(* IEC 61131-3 sources: myCodes/Stone/07.02.2022 - OOPs Approach/MPx_One_New/Mpx_One_Source_Code/MPx_One/3. USHPXMPX010A1/USHPXMPX010A1/MPXone_Medium/DFR_Libs (part 2) *)

/// Light Function ///

FUNCTION_BLOCK DFR_DiagLights
    VAR_INPUT
        Inp : BOOL;
        TotTime : REAL;
    END_VAR
    VAR_OUTPUT
        Out : BOOL;
        TimerDone : BOOL;
    END_VAR
    VAR
        LightTimer : DFRTimer;
    END_VAR
    IF Inp THEN
        LightTimer(Ena := Inp, PLCCycletime := 0.5, ProgramTime := TotTime);
        IF LightTimer.ElapsedTime <= (TotTime / 10) THEN
            Out := TRUE;
        ELSIF LightTimer.ElapsedTime > (TotTime / 10) AND LightTimer.ElapsedTime <= (TotTime / 7.5) THEN
            Out := FALSE;
        ELSIF LightTimer.ElapsedTime > (TotTime / 7.5) AND LightTimer.ElapsedTime <= (TotTime / 5) THEN
            Out := TRUE;
        ELSIF LightTimer.ElapsedTime > (TotTime / 5) AND LightTimer.ElapsedTime <= (TotTime / 2.5) THEN
            Out := FALSE;
        ELSIF LightTimer.ElapsedTime > (TotTime / 2.5) AND LightTimer.ElapsedTime <= (TotTime / 2) THEN
            Out := TRUE;
        ELSIF LightTimer.ElapsedTime > (TotTime / 2) AND LightTimer.ElapsedTime <= (TotTime / 1.5) THEN
            Out := FALSE;
        ELSIF LightTimer.ElapsedTime > (TotTime / 1.5) AND LightTimer.ElapsedTime <= (TotTime / 1.25) THEN
            Out := TRUE;
        ELSE
            Out := FALSE;
        END_IF;
        IF LightTimer.Q THEN
            LightTimer(Ena := FALSE);
            TimerDone := TRUE;
        END_IF;
    ELSE
        Out := FALSE;
        TimerDone := FALSE;
        LightTimer(Ena := FALSE);

    END_IF;
END_FUNCTION_BLOCK

/// ************  EOL Run Test Functions ************///

/// EOL Pull Down Test Function ///

FUNCTION_BLOCK DFR_Feature_PullDownTest
    VAR_INPUT
        Enable             : BOOL; // To Enable the Regulation
        CycleTime          : REAL; // To change the Cycle Time of the Pull Down Test Function
        Preset_RegTime     : REAL; // Regulation Timer
        Preset_RegFailTime : REAL; // Regulation Fail Timer
        Preset_WaitTime    : REAL; // Regulation Wait Timer
        In1                : REAL; // Discharge Air Temp
        In2                : REAL; // Defrost Temp
        Reg_SP             : REAL; // Regulation Setpoint
        FanSP              : REAL; // Fan Setpoint
        FanHystSP          : REAL; // Fan Hysterisis SP

    END_VAR
    VAR
        Reg_Fail_Timer     : DFRTimer; // Enable the Fail Timer if Discharge Air Temp fails to meet the SP
        RegulationTimer    : DFRTimer; // Enable Regulation Timer to monitor Discharge Air temp

    END_VAR
    VAR_OUTPUT
        DFR_Regulation_Sts : STRING; // DFR Regulation Test Status
        Out1               : BOOL; // CDU Enable - V_OM_Solenoid_Flag
        Out2               : BOOL; // Fan Enable - V_OM_Fans_Flag
    END_VAR

    IF Enable AND (V_CSM_EOL_Test_Result = 0 OR V_CSM_EOL_Test_Result = 3) THEN
        Out1 := TRUE;
        IF In1 <= Reg_SP THEN
            RegulationTimer(Ena := TRUE, PLCCycletime := CycleTime, ProgramTime := Preset_RegTime);
            Reg_Fail_Timer(Ena := FALSE);
            IF RegulationTimer.Q THEN
                DFR_Regulation_Sts := 'PAS';
                RegulationTimer(Ena := FALSE);
            END_IF;
        ELSE
            Reg_Fail_Timer(Ena := TRUE, PLCCycletime := CycleTime, ProgramTime := Preset_RegFailTime);
            RegulationTimer(Ena := FALSE);
            IF Reg_Fail_Timer.Q THEN
                DFR_Regulation_Sts := 'FAL';
                Reg_Fail_Timer(Ena := FALSE);
            END_IF;
        END_IF;

        IF  (DFR_CINCaseSystemComponent(6) = 0) OR (DFR_CINCaseSystemComponent(9) = 2) THEN // No Door Case and MT Case
            Out2 := TRUE;
        ELSIF (NOT (DFR_CINCaseSystemComponent(6) = 0) AND (DFR_CINCaseSystemComponent(9) = 1)) THEN // LT Door Case Only
            IF In2 <= FanSP THEN // Fans will be turned On if Defrost Temp is less than Fan Setpoint
                Out2 := TRUE;
            ELSIF In2 > FanSP + FanHystSP THEN
                Out2 := FALSE;
            END_IF;
        ELSE
            Out2 := FALSE;
        END_IF;
    ELSIF (DFR_Regulation_Sts = 'FAL') OR(DFR_Regulation_Sts = 'PAS') THEN
        RegulationTimer(Ena := FALSE);
        Reg_Fail_Timer(Ena := FALSE);
    END_IF;
END_FUNCTION_BLOCK

/// Defrost Cycle Test Function  ///

FUNCTION_BLOCK DFR_Feature_DefrostCycleTest
    VAR_INPUT
        Enable : BOOL;       // To Enable the Defrost Cycle Test
        CycleTime : REAL;
        Preset_DefFailTime : REAL;
        In1 : REAL; // Defrost Termination Temperature OR Discharge Air Temp (If Defrost Probe is absent)
        SetPoint : REAL;  // Defrost Termination Temperature SP

    END_VAR
    VAR
        Def_Fail_Timer : DFRTimer; // Enable the Fail Timer if change in Defrost Term Temp fails to meet the SP
        TempDelta : REAL;
        PrevIn : REAL;
        SaveFlag : bool := FALSE;
    END_VAR

    VAR_OUTPUT
        DFR_DefrostCycle_Sts : STRING; // DFR Defrost Cycle Test Status
        Out1 : BOOL; // CDU Disable - V_OM_Solenoid_Flag
        Out2 : BOOL; // Defrost Enable - V_OM_Defrost_Flag
        Out3 : BOOL; // Fan Disable - V_OM_Fans_Flag
        Out4 : BOOL; // Drain Heater - V_OM_DrainHeat_Flag
    END_VAR

    Def_Fail_Timer(Ena := Enable, PLCCycletime := CycleTime, ProgramTime := Preset_DefFailTime);
    IF Enable AND (V_CSM_EOL_Test_Result = 0 OR V_CSM_EOL_Test_Result = 3) THEN
        IF(NOT SaveFlag) THEN
            SaveFlag := TRUE;
            //PrevIn := In1;
        //ELSE
            //TempDelta := (In1 - PrevIn); // Discharge Air Temp difference
        END_IF;

        Out2 := TRUE; // Defrost Should be Enabled
        Out1 := FALSE; // CDU should be Disabled
        IF Out2 AND NOT Out1 THEN
            IF In1 > Setpoint THEN
                Def_Fail_Timer(Ena := FALSE);
                DFR_DefrostCycle_Sts := 'PAS';
            ELSE
                ;
            END_IF;
        END_IF;

        IF Def_Fail_Timer.Q THEN
            DFR_DefrostCycle_Sts := 'FAL';
            Def_Fail_Timer(Ena := FALSE);
        END_IF;

        IF  (DFR_CINCaseSystemComponent(6) = 0) OR (DFR_CINCaseSystemComponent(9) = 2) THEN // No Door Case and MT Case
            Out3 := TRUE; // Fans are ON
            Out4 := FALSE; // Drain Heater are Disabled
        ELSIF (NOT (DFR_CINCaseSystemComponent(6) = 0) AND (DFR_CINCaseSystemComponent(9) = 1)) THEN // LT Door Case Only
            Out3 := FALSE; // Fans are OFF
            Out4 := TRUE; // Drain Heater are Enabled
        ELSE
            Out3 := FALSE; // Fans are OFF
            Out4 := FALSE; // Drain Heater are Disabled
        END_IF;
    ELSE
        PrevIn := In1;
        TempDelta := 0;
        SaveFlag := FALSE;
        DFR_DefrostCycle_Sts := 'NA';
        Def_Fail_Timer(Ena := FALSE);
    END_IF;

END_FUNCTION_BLOCK
/*
FUNCTION_BLOCK DFR_MOV_AVERAGE
    VAR_INPUT
        in_sample : real;
        in_count  : uint := 1; //It should be less than total no. of array samples
    END_VAR

    VAR
        array_real : ARRAY[1..64] OF real;
        sum        : real;
        index      : uint := 1;
    END_VAR

    VAR_OUTPUT
        out_mean : real;
    END_VAR

    sum := sum - array_real[index] + in_sample;
    array_real[index] := in_sample;
    index := index + 1;

    IF(index >= in_count) THEN
        index := 1;
    END_IF;

    out_mean := sum / UINT_TO_REAL(in_count);
END_FUNCTION_BLOCK
*/
FUNCTION_BLOCK DFR_FB_CompressorProtection
    VAR_INPUT
        in_CompressorStatus         : BOOL;
        in_T1Mins                   : USINT     := 60;
        in_T2Mins                   : USINT     := 5;
        in_Count1                   : USINT     := 2;
        in_Count2                   : USINT     := 4;
        in_Reset                    : BOOL      := FALSE;
        in_CompShutdownOn           : BOOL      := FALSE;
    END_VAR
    VAR_OUTPUT
        out_ShutdownCommand         : BOOL      := FALSE;
        out_WarningLow              : BOOL      := FALSE;
        out_WarningMedium           : BOOL      := FALSE;
        out_WarningSevere           : BOOL      := FALSE;
    END_VAR
    VAR
        fb_Timer1                   : TON;
        fb_Timer2                   : TON;
        fb_FTrig1                   : F_TRIG;
        fb_RTrig1                   : R_TRIG;
        b_init                      : BOOL           := FALSE;
        b_EnableTimer1              : BOOL           := FALSE;
        b_EnableTimer2              : BOOL           := FALSE;
        n_Counter                   : USINT          := 0;
    END_VAR
    {REGION INIT}
    IF (NOT b_init) THEN
        fb_Timer1.PT                := to_time(in_T1Mins) * (60 * 1000);    // minutes to milli-seconds
        fb_Timer2.PT                := to_time(in_T2Mins) * (60 * 1000);
        out_ShutdownCommand         := FALSE;
        out_WarningLow              := FALSE;
        out_WarningMedium           := FALSE;
        out_WarningSevere           := FALSE;
        b_init                      := TRUE;
    ELSE
    END_IF;
    {ENDREGION}
    {REGION RESET LOGIC}
    fb_RTrig1(CLK := in_Reset);
    IF fb_RTrig1.Q THEN
        n_Counter := 0;
        fb_Timer1(IN    := FALSE);
        fb_Timer2(IN    := FALSE);
        fb_FTrig1(CLK   := FALSE);
        out_ShutdownCommand         := FALSE;
        out_WarningLow              := FALSE;
        out_WarningMedium           := FALSE;
        out_WarningSevere           := FALSE;
    ELSE
    END_IF;
    {ENDREGION}
    {REGION FALL COUNT}
    fb_FTrig1(CLK := in_CompressorStatus);
    IF fb_FTrig1.Q THEN
        n_Counter           := n_Counter + 1;
        IF(n_Counter = 1) THEN
            b_EnableTimer1      := TRUE;
        ELSE
        END_IF;
    END_IF;

    fb_Timer1(IN := b_EnableTimer1);

    IF fb_Timer1.Q THEN
        n_Counter           := 0;
        b_EnableTimer1      := FALSE;
    ELSE
    END_IF;

    IF (n_Counter < in_Count1) THEN
        out_WarningLow          := FALSE;
    ELSIF (n_Counter >= in_Count1) AND (n_Counter < in_Count2) THEN
        out_WarningLow          := TRUE;
    ELSIF(n_Counter >= in_Count2) THEN
        out_WarningSevere       := TRUE;
        out_ShutdownCommand     := in_CompShutdownOn;
    ELSE
    END_IF;
    {ENDREGION}
    {REGION DURATION}
    b_EnableTimer2 := NOT (in_CompressorStatus);
    fb_Timer2(IN := b_EnableTimer2);
    IF (fb_Timer2.Q) THEN
        out_WarningMedium   := TRUE;
    ELSE
        out_WarningMedium   := FALSE;
    END_IF;
    {ENDREGION}
END_FUNCTION_BLOCK

FUNCTION DFR_F_Bitpacking : INT
    VAR_INPUT
        in : ARRAY[0..15] OF BOOL;
    END_VAR

    VAR
        i : INT;
        b : REAL := 2;
    END_VAR
    DFR_F_Bitpacking := 0;
    FOR i := 0 TO 15 DO
        DFR_F_Bitpacking := DFR_F_Bitpacking + TO_INT(expt(b, i)) * TO_INT(in[i]);
    END_FOR;

END_FUNCTION

TYPE
    U_BITPACK : UNION
        arr : ARRAY[0..15] OF bool;
        i : UINT;
    END_UNION;
END_TYPE

TYPE
    T_SP_SYSTEM : STRUCT
        info           : U_BITPACK;
        alarm          : U_BITPACK;
        alarmflag      : BOOL;
        infoflag       : BOOL;
    END_STRUCT;
END_TYPE

TYPE
    T_SP_HPX : STRUCT
        system   : T_SP_SYSTEM;
        comp     : T_SP_SYSTEM;
        cond     : T_SP_SYSTEM;
        evap     : T_SP_SYSTEM;
        metering : T_SP_SYSTEM;
        comm     : T_SP_SYSTEM;
        device   : T_SP_SYSTEM;
    END_STRUCT;
END_TYPE

FUNCTION_BLOCK DFR_FB_Blinker
    VAR_INPUT
        InSignal : bool := FALSE;
        DelaySecs : int := 60;
        Count : int := 2;
    END_VAR

    VAR_OUTPUT
        Out : bool := FALSE;
    END_VAR

    VAR
        OnDelay : ton;
        OnPulse : tp;
        OutCount : r_trig;
        InRise : r_trig;
        OutEnable : bool := FALSE;
        Counter : int := 0;
    END_VAR

    OnDelay.PT := to_time(DelaySecs) * 1000;    // seconds to milliseconds
    OnPulse.PT := to_time(DelaySecs) * 1000;

    InRise(CLK := InSignal);
    IF(InRise.Q) THEN
        Counter := 0;
        OutEnable := TRUE;
    ELSE
    END_IF;

    OutCount(CLK := Out);
    IF(OutCount.Q) THEN
        Counter := Counter + 1;
    ELSE
    END_IF;

    IF(Counter >= Count) THEN
        OutEnable := FALSE;
    ELSE
    END_IF;

    OnDelay(IN := (InSignal AND NOT OnPulse.Q AND OutEnable));
    OnPulse(IN := OnDelay.Q);

    Out := NOT(OnPulse.Q);
END_FUNCTION_BLOCK

FUNCTION WizDone_Action : REAL;
END_FUNCTION

FUNCTION_BLOCK DFR_EnterProg
    VAR_INPUT
        In : BOOL;
    END_VAR
    IF In THEN
        En_GlobalSwitch_Override  := TRUE;
        En_DrainHeaterOverwrite   := TRUE;
        En_RailHeaterOverwrite    := TRUE;
        En_LightOverwrite         := TRUE;
        En_FansOverwrite          := TRUE;
        En_FansModulOverwrite     := TRUE;
        En_ValveModulOverwrite    := TRUE;
        En_HeatersModulOverwrite  := TRUE;
    END_IF;

END_FUNCTION_BLOCK

FUNCTION_BLOCK DFR_DrainHeater_Enable
    VAR_INPUT
        In : BOOL;
    END_VAR
    IF In THEN
        En_GlobalSwitch_Override := TRUE;
        En_DrainHeaterOverwrite := TRUE;
    ELSE
        En_DrainHeaterOverwrite := FALSE;
    END_IF;

END_FUNCTION_BLOCK

FUNCTION_BLOCK DFR_RailHeater_Enable
    VAR_INPUT
        In : BOOL;
    END_VAR
    IF In THEN
        En_GlobalSwitch_Override := TRUE;
        En_RailHeaterOverwrite   := TRUE;
        En_HeatersModulOverwrite := TRUE;
    ELSE
        En_RailHeaterOverwrite   := FALSE;
        En_HeatersModulOverwrite := FALSE;
    END_IF;

END_FUNCTION_BLOCK

FUNCTION_BLOCK DFR_Lights_Enable
    VAR_INPUT
        In : BOOL;
    END_VAR
    IF In THEN
        En_GlobalSwitch_Override := TRUE;
        En_LightOverwrite        := TRUE;
    ELSE
        En_LightOverwrite        := FALSE;
    END_IF;

END_FUNCTION_BLOCK

FUNCTION_BLOCK DFR_Fans_Enable
    VAR_INPUT
        In : BOOL;
    END_VAR
    IF In THEN
        En_GlobalSwitch_Override := TRUE;
        En_FansOverwrite         := TRUE;
        En_FansModulOverwrite    := TRUE;
    ELSE
        En_FansOverwrite      := FALSE;
        En_FansModulOverwrite := FALSE;
    END_IF;

END_FUNCTION_BLOCK

FUNCTION_BLOCK DFR_EEV_Enable
    VAR_INPUT
        In : BOOL;
    END_VAR
    IF In THEN
        En_GlobalSwitch_Override := TRUE;
        En_ValveModulOverwrite   := TRUE;
    ELSE
        En_ValveModulOverwrite   := FALSE;
    END_IF;

END_FUNCTION_BLOCK

(* ---- DFR_Utility_Class.st ---- *)
USING System.Math;
USING System;
USING System.Timer;
USING System.Text;

CLASS PUBLIC DFR_LIBRARY
    (**
    This class library contains majorly used
    functions required for development
    of the Dover Food and Retail Case Platform.

    Initial Development: Rohit Maity
                         08/01/2022
    **)

    METHOD PUBLIC DFR_DiagAntiSweatHeater

        VAR_INPUT
            Inp : BOOL;
            Trigger : BOOL;
          //TotTime : REAL;
        END_VAR

        VAR_IN_OUT
            Out1 : BOOL;
            Out2 : REAL;
          //TimerDone : BOOL;
            Test_Status : STRING;
        END_VAR

    IF Inp AND NOT Trigger THEN
        Out1 := TRUE;
        Out2 := 100;
        Test_Status := 'NA';
    ELSIF (Inp AND Trigger) THEN
        Out1 := FALSE;
        Out2 := 0;
        Test_Status := 'PAS';
    END_IF;

    END_METHOD

    METHOD PUBLIC DFR_DiagLights

    VAR_INPUT
        Inp : BOOL;
        TotTime : REAL;
    END_VAR

    VAR_IN_OUT
        Out : BOOL;
        TimerDone : BOOL;
    END_VAR

    VAR
        LightTimer : DFRTimer;
    END_VAR

    IF Inp THEN
        LightTimer(Ena := Inp, PLCCycletime := 0.5, ProgramTime := TotTime);
        IF LightTimer.ElapsedTime <= (TotTime / 10) THEN
            Out := TRUE;
        ELSIF LightTimer.ElapsedTime > (TotTime / 10) AND LightTimer.ElapsedTime <= (TotTime / 7.5) THEN
            Out := FALSE;
        ELSIF LightTimer.ElapsedTime > (TotTime / 7.5) AND LightTimer.ElapsedTime <= (TotTime / 5) THEN
            Out := TRUE;
        ELSIF LightTimer.ElapsedTime > (TotTime / 5) AND LightTimer.ElapsedTime <= (TotTime / 2.5) THEN
            Out := FALSE;
        ELSIF LightTimer.ElapsedTime > (TotTime / 2.5) AND LightTimer.ElapsedTime <= (TotTime / 2) THEN
            Out := TRUE;
        ELSIF LightTimer.ElapsedTime > (TotTime / 2) AND LightTimer.ElapsedTime <= (TotTime / 1.5) THEN
            Out := FALSE;
        ELSIF LightTimer.ElapsedTime > (TotTime / 1.5) AND LightTimer.ElapsedTime <= (TotTime / 1.25) THEN
            Out := TRUE;
        ELSE
            Out := FALSE;
        END_IF;
        IF LightTimer.Q THEN
            LightTimer(Ena := FALSE);
            TimerDone := TRUE;
        END_IF;
    ELSE
        Out := FALSE;
        TimerDone := FALSE;
        LightTimer(Ena := FALSE);

    END_IF;
    END_METHOD

    METHOD PUBLIC DFR_DiagDrainheater
        VAR_INPUT
        Inp : BOOL;
        Trigger : BOOL;
        //TotTime : REAL;
    END_VAR

    VAR
        //DrainHtrTimer : DFRTimer;
    END_VAR
    VAR_IN_OUT
        Output : BOOL;
        //TimerDone : BOOL;
        Test_Status : STRING;
    END_VAR
    IF Inp AND NOT Trigger THEN
        Output := TRUE;
        Test_Status := 'NA';
    ELSIF (Inp AND Trigger) THEN
        Output := FALSE;
        Test_Status := 'PAS';
    END_IF;

    END_METHOD

    METHOD PUBLIC DFR_CINCaseSystemComponent:INT
        VAR_INPUT
        comp_num : INT;
        END_VAR
    VAR
        out_info    : string;
        length      : int;
        str1        : string;
        str2        : string;
        str3        : string;
        str4        : string;
        str5        : string;
        str6        : string;
    END_VAR

  //  V_CSM_CaseSystemInfo := '05052021121065001113237';

    str1 := format('%04u', C_CSM_CaseSystemInfo1);
    str2 := format('%04u', C_CSM_CaseSystemInfo2);
    str3 := format('%04u', C_CSM_CaseSystemInfo3);
    str4 := format('%04u', C_CSM_CaseSystemInfo4);
    str5 := format('%04u', C_CSM_CaseSystemInfo5);
    str6 := format('%03u', C_CSM_CaseSystemInfo6);

    V_CSM_CaseSystemInfo := str1 + str2 + str3 + str4 + str5 + str6;

    length := to_int(len(V_CSM_CaseSystemInfo));

    IF length <= 1 AND NOT WIZDONE THEN
        V_CSM_InvalidCIN_Flag := TRUE;
        out_info := '0';
    ELSE
         V_CSM_InvalidCIN_Flag := FALSE;
        CASE comp_num OF
            1: // Case date
                out_info := left(V_CSM_CaseSystemInfo, 2);
            2: // Case month
                out_info := mid(V_CSM_CaseSystemInfo, 2, 2);
            3: // Case year
                out_info := mid(V_CSM_CaseSystemInfo, 4, 4);
            4: // Case Series
                out_info := mid(V_CSM_CaseSystemInfo, 3, 8);
            5: // Refrigerant : 1-R-22, 2-R-404A, 3-R-407A, 4-R-410A, 5-R-422D, 6-R-507A, 7-R-448A, 8-R-449A, 9-CO2 DX, 10-CO2 SC, 11-Glycol SC
                out_info := mid(V_CSM_CaseSystemInfo, 2, 11);
            6: // Doors : 0,1,2,3,4,5,6
                out_info := mid(V_CSM_CaseSystemInfo, 1, 13);
            7: // Length in feet : 0,4,6,8,10,12
                out_info := mid(V_CSM_CaseSystemInfo, 2, 14);
            8: // Evaporator : 0-Standard , 1- NRG
                out_info := mid(V_CSM_CaseSystemInfo, 1, 16);
            9: // Control Temp : 0 -Dual,1-LT ,2-MT
                out_info := mid(V_CSM_CaseSystemInfo, 1, 17);
            10: // Defrost Type : 0-Off-time, 1-Electric, 2-Hotgas
                out_info := mid(V_CSM_CaseSystemInfo, 1, 18);
            11: // Metering Device Type : 0-None, 1-TXV, 2-PWM, 3-Stepper
                out_info := mid(V_CSM_CaseSystemInfo, 1, 19);
            12: // Temperature Control Type : 1-Self Contained, 2-Remote
                out_info := mid(V_CSM_CaseSystemInfo, 1, 20);
            13: // Controller Type : 1- Dixell, 2- MPXOne, 3 – Cpco Mini
                out_info := mid(V_CSM_CaseSystemInfo, 2, 21);
            ELSE
                out_info := '0';
        END_CASE;
    END_IF;
    DFR_CINCaseSystemComponent := to_int(out_info);

        END_METHOD

END_CLASS

CLASS PUBLIC UnitTestingAssertions
(**

    Initial Creation:
    09/02/2022
    Rohit Maity

    This has been created to make Automatic Testing on Results from Function Blocks created for DFR.

*)

    VAR PUBLIC

    END_VAR

    VAR

    END_VAR

    (**
    Timer Initial Methods called Init
    **)

    METHOD Init

    END_METHOD

   (**
                 Testing INT Equality
    **)

    METHOD assertEquals

        VAR_INPUT
            IN : BOOL;
            intActualResult : INT;
            intExpectedResult : INT;

        END_VAR

        VAR_IN_OUT
            Status : STRING;

        END_VAR

        VAR
            Output : INT;
            OneShot : R_TRIG;
        END_VAR

        OneShot(CLK := IN);

    IF (OneShot.Q) THEN
        IF  (intActualResult = intExpectedResult) THEN

                Output := 1;

        ELSIF (intActualResult <> intExpectedResult) THEN
               Output := 2;

        ELSIF (NOT IN) AND (Output<>0) THEN
                //Output := 0;

        END_IF;

    END_IF;

    CASE Output OF
        0: Status := 'The Test is not Running';
        1: Status := 'PASSED';
        2: Status := 'FAILED';
        4: Status := 'Test is Running';
    END_CASE;

    END_METHOD

    (**
            Testing REAL Equality
    **)

    METHOD assertEquals

        VAR_INPUT
            IN : BOOL;
            realActualResult : REAL;
            realExpectedResult : REAL;
        END_VAR

        VAR_IN_OUT
            Status : STRING;
        END_VAR

        VAR
            Output : INT;
            OneShot : R_TRIG;
        END_VAR

        OneShot(CLK := IN);

    IF (OneShot.Q) THEN
        IF  (realActualResult = realExpectedResult) THEN
                Output := 1;

        ELSIF (realActualResult <> realExpectedResult) THEN

               Output := 2;

        ELSIF (NOT IN) AND (Output<>0) THEN
                //Output := 0;

        END_IF;

    END_IF;

    CASE Output OF
        0: Status := 'The Test is not Running';
        1: Status := 'PASSED';
        2: Status := 'FAILED';
        4: Status := 'Test is Running';
    END_CASE;

    END_METHOD

    (**
           Testing BOOLEAN Equality
    **)

    METHOD assertEquals

        VAR_INPUT
            IN : BOOL;
            boolActualResult :BOOL;
            boolExpectedResult : BOOL;

        END_VAR

        VAR_IN_OUT
            Status : STRING;
        END_VAR

        VAR
            Output : INT;
            OneShot : R_TRIG;
        END_VAR

        OneShot(CLK := IN);

    IF (OneShot.Q) THEN
        IF  (boolActualResult = boolExpectedResult) THEN

                Output := 1;

        ELSIF (boolActualResult <> boolExpectedResult) THEN

               Output := 2;

        ELSIF (NOT IN) AND (Output<>0) THEN
                //Output := 0;

        END_IF;

    END_IF;

    CASE Output OF
        0: Status := 'The Test is not Running';
        1: Status := 'PASSED';
        2: Status := 'FAILED';
        4: Status := 'Test is Running';
    END_CASE;

    END_METHOD

    METHOD assertEquals

        VAR_INPUT
            IN : BOOL;
            stringActualResult :  STRING;
            stringExpectedResult : STRING;
        END_VAR

        VAR_IN_OUT
            Status : STRING;
        END_VAR

        VAR
            Output : INT;
            OneShot : R_TRIG;
        END_VAR

        OneShot(CLK := IN);

    IF (OneShot.Q) THEN
        IF  (stringActualResult = stringExpectedResult) THEN

                Output := 1;

        ELSIF (stringActualResult <> stringExpectedResult) THEN

               Output := 2;

        ELSIF (NOT IN) AND (Output<>0) THEN
                //Output := 0;
        END_IF;

    END_IF;

    CASE Output OF
        0: Status := 'The Test is not Running';
        1: Status := 'PASSED';
        2: Status := 'FAILED';
        4: Status := 'Test is Running';
    END_CASE;

    END_METHOD

    METHOD assertTrue
        (*
        This Test
        *)

        VAR_INPUT
            IN : BOOL;
            actualResult : BOOL;
        END_VAR

        VAR_IN_OUT
            Status : STRING;
        END_VAR

        VAR
            Output : INT;
            OneShot : R_TRIG;
        END_VAR

        OneShot(CLK := IN);

    IF (OneShot.Q) THEN
        IF  (actualResult = TRUE) THEN

                Output := 1;

        ELSIF (actualResult = FALSE) THEN

               Output := 2;

        ELSIF (NOT IN) AND (Output<>0) THEN
                //Output := 0;

        END_IF;

    END_IF;

    CASE Output OF
        0: Status := 'The Test is not Running';
        1: Status := 'PASSED';
        2: Status := 'FAILED';
        4: Status := 'Test is Running';
    END_CASE;

END_METHOD

    METHOD assertFalse

        VAR_INPUT
            IN : BOOL;
            actualResult : BOOL;
        END_VAR

        VAR_IN_OUT
            Status : STRING;
        END_VAR

        VAR
            Output : INT;
            OneShot : R_TRIG;
        END_VAR

        OneShot(CLK := IN);

    IF (OneShot.Q) THEN
        IF  (actualResult = FALSE) THEN

                Output := 1;

        ELSIF (actualResult = TRUE) THEN

                Output := 2;

        ELSIF (NOT IN) AND (Output<>0) THEN
                //Output := 0;

        END_IF;

    END_IF;

    CASE Output OF
        0: Status := 'The Test is not Running';
        1: Status := 'PASSED';
        2: Status := 'FAILED';
        4: Status := 'Test is Running';
    END_CASE;

END_METHOD

END_CLASS

CLASS PUBLIC STUnit EXTENDS UnitTestingAssertions

    VAR
      Enable : BOOL;
    END_VAR

    METHOD InitializeTests

    END_METHOD

    METHOD RunAllTests

        Enable := TRUE;

    END_METHOD

    METHOD BeforeTest

    END_METHOD

    METHOD AfterTest

        Enable := FALSE;

    END_METHOD

    METHOD TestMethod

    END_METHOD

    METHOD TestInstance

        VAR_INPUT
           TestMode: STRING;
        END_VAR

        IF(Enable) THEN
            IF(TestMode='Before') THEN
            BeforeTest();
            ELSIF (TestMode='After') THEN
            AfterTest();
            ELSIF (TestMode='TestMethod') THEN
            AfterTest();
            ELSE

            END_IF;
        END_IF;

    END_METHOD

END_CLASS

(* ---- DFR_Utility_v1.st ---- *)
USING System.Math;
USING System;
USING System.Timer;
USING System.Text;

CLASS PUBLIC DFR_LIBRARY
    (**
    This class library contains majorly used
    functions required for development
    of the Dover Food and Retail Case Platform.

    Initial Development: Rohit Maity
                         08/01/2022
    **)

    METHOD PUBLIC DFR_DiagAntiSweatHeater

        VAR_INPUT
            Inp : BOOL;
            Trigger : BOOL;
          //TotTime : REAL;
        END_VAR

        VAR_IN_OUT
            Out1 : BOOL;
            Out2 : REAL;
          //TimerDone : BOOL;
            Test_Status : STRING;
        END_VAR

    IF Inp AND NOT Trigger THEN
        Out1 := TRUE;
        Out2 := 100;
        Test_Status := 'NA';
    ELSIF (Inp AND Trigger) THEN
        Out1 := FALSE;
        Out2 := 0;
        Test_Status := 'PAS';
    END_IF;

    END_METHOD

    METHOD PUBLIC DFR_DiagLights

    VAR_INPUT
        Inp : BOOL;
        TotTime : REAL;
    END_VAR

    VAR_IN_OUT
        Out : BOOL;
        TimerDone : BOOL;
    END_VAR

    VAR
        LightTimer : DFRTimer;
    END_VAR

    IF Inp THEN
        LightTimer(Ena := Inp, PLCCycletime := 0.5, ProgramTime := TotTime);
        IF LightTimer.ElapsedTime <= (TotTime / 10) THEN
            Out := TRUE;
        ELSIF LightTimer.ElapsedTime > (TotTime / 10) AND LightTimer.ElapsedTime <= (TotTime / 7.5) THEN
            Out := FALSE;
        ELSIF LightTimer.ElapsedTime > (TotTime / 7.5) AND LightTimer.ElapsedTime <= (TotTime / 5) THEN
            Out := TRUE;
        ELSIF LightTimer.ElapsedTime > (TotTime / 5) AND LightTimer.ElapsedTime <= (TotTime / 2.5) THEN
            Out := FALSE;
        ELSIF LightTimer.ElapsedTime > (TotTime / 2.5) AND LightTimer.ElapsedTime <= (TotTime / 2) THEN
            Out := TRUE;
        ELSIF LightTimer.ElapsedTime > (TotTime / 2) AND LightTimer.ElapsedTime <= (TotTime / 1.5) THEN
            Out := FALSE;
        ELSIF LightTimer.ElapsedTime > (TotTime / 1.5) AND LightTimer.ElapsedTime <= (TotTime / 1.25) THEN
            Out := TRUE;
        ELSE
            Out := FALSE;
        END_IF;
        IF LightTimer.Q THEN
            LightTimer(Ena := FALSE);
            TimerDone := TRUE;
        END_IF;
    ELSE
        Out := FALSE;
        TimerDone := FALSE;
        LightTimer(Ena := FALSE);

    END_IF;
    END_METHOD

    METHOD PUBLIC DFR_DiagDrainheater
        VAR_INPUT
        Inp : BOOL;
        Trigger : BOOL;
        //TotTime : REAL;
    END_VAR

    VAR
        //DrainHtrTimer : DFRTimer;
    END_VAR
    VAR_IN_OUT
        Output : BOOL;
        //TimerDone : BOOL;
        Test_Status : STRING;
    END_VAR
    IF Inp AND NOT Trigger THEN
        Output := TRUE;
        Test_Status := 'NA';
    ELSIF (Inp AND Trigger) THEN
        Output := FALSE;
        Test_Status := 'PAS';
    END_IF;

    END_METHOD

    METHOD PUBLIC DFR_CINCaseSystemComponent:INT
        VAR_INPUT
        comp_num : INT;
        END_VAR
    VAR
        out_info    : string;
        length      : int;
        str1        : string;
        str2        : string;
        str3        : string;
        str4        : string;
        str5        : string;
        str6        : string;
    END_VAR

  //  V_CSM_CaseSystemInfo := '05052021121065001113237';

    str1 := format('%04u', C_CSM_CaseSystemInfo1);
    str2 := format('%04u', C_CSM_CaseSystemInfo2);
    str3 := format('%04u', C_CSM_CaseSystemInfo3);
    str4 := format('%04u', C_CSM_CaseSystemInfo4);
    str5 := format('%04u', C_CSM_CaseSystemInfo5);
    str6 := format('%03u', C_CSM_CaseSystemInfo6);

    V_CSM_CaseSystemInfo := str1 + str2 + str3 + str4 + str5 + str6;

    length := to_int(len(V_CSM_CaseSystemInfo));

    IF length <= 1 AND NOT WIZDONE THEN
        V_CSM_InvalidCIN_Flag := TRUE;
        out_info := '0';
    ELSE
         V_CSM_InvalidCIN_Flag := FALSE;
        CASE comp_num OF
            1: // Case date
                out_info := left(V_CSM_CaseSystemInfo, 2);
            2: // Case month
                out_info := mid(V_CSM_CaseSystemInfo, 2, 2);
            3: // Case year
                out_info := mid(V_CSM_CaseSystemInfo, 4, 4);
            4: // Case Series
                out_info := mid(V_CSM_CaseSystemInfo, 3, 8);
            5: // Refrigerant : 1-R-22, 2-R-404A, 3-R-407A, 4-R-410A, 5-R-422D, 6-R-507A, 7-R-448A, 8-R-449A, 9-CO2 DX, 10-CO2 SC, 11-Glycol SC
                out_info := mid(V_CSM_CaseSystemInfo, 2, 11);
            6: // Doors : 0,1,2,3,4,5,6
                out_info := mid(V_CSM_CaseSystemInfo, 1, 13);
            7: // Length in feet : 0,4,6,8,10,12
                out_info := mid(V_CSM_CaseSystemInfo, 2, 14);
            8: // Evaporator : 0-Standard , 1- NRG
                out_info := mid(V_CSM_CaseSystemInfo, 1, 16);
            9: // Control Temp : 0 -Dual,1-LT ,2-MT
                out_info := mid(V_CSM_CaseSystemInfo, 1, 17);
            10: // Defrost Type : 0-Off-time, 1-Electric, 2-Hotgas
                out_info := mid(V_CSM_CaseSystemInfo, 1, 18);
            11: // Metering Device Type : 0-None, 1-TXV, 2-PWM, 3-Stepper
                out_info := mid(V_CSM_CaseSystemInfo, 1, 19);
            12: // Temperature Control Type : 1-Self Contained, 2-Remote
                out_info := mid(V_CSM_CaseSystemInfo, 1, 20);
            13: // Controller Type : 1- Dixell, 2- MPXOne, 3 – Cpco Mini
                out_info := mid(V_CSM_CaseSystemInfo, 2, 21);
            ELSE
                out_info := '0';
        END_CASE;
    END_IF;
    DFR_CINCaseSystemComponent := to_int(out_info);

        END_METHOD

END_CLASS

CLASS PUBLIC UnitTesting
(**

    Initial Creation:
    09/02/2022
    DFR Control

    This has been created to make Automatic Testing on Results from Function Blocks created for DFR.

**)

    VAR PUBLIC
        PassTimeSP : TIME;
        FailTimeSP : TIME;
    END_VAR

    VAR
       PassTimer : TON;
       FailTimer : TON;
    END_VAR

    (**
    Timer Initial Methods called Init
    **)

    METHOD Init
        PassTimer(PT := PassTimeSP);
        FailTimer(PT := FailTimeSP);
    END_METHOD

   (**
                 Testing INT Equality
    **)

    METHOD assertEquals

        VAR_INPUT
            IN : BOOL;
            intActualResult : INT;
            intExpectedResult : INT;

        END_VAR

        VAR_IN_OUT
            Status : STRING;

        END_VAR

        VAR
            Output : INT;
        END_VAR

        Init();

    IF (IN) THEN
        IF  (intActualResult = intExpectedResult) THEN
            PassTimer.IN := TRUE;

            IF(NOT PassTimer.Q) THEN
                Output := 4;
            END_IF;

            IF(PassTimer.Q) THEN
                Output := 1;
                PassTimer.IN := FALSE;

            END_IF;

        ELSIF (intActualResult <> intExpectedResult) THEN
            FailTimer(In := TRUE);

            IF(NOT FailTimer.Q) THEN
                Output := 4;
            END_IF;

            IF(FailTimer.Q) THEN
               Output := 2;
               FailTimer.In := FALSE;

            END_IF;
        END_IF;
    ELSIF (NOT IN) AND (Output<>0) THEN
                //Output := 0;

    END_IF;

    CASE Output OF
        0: Status := 'The Test is not Running';
        1: Status := 'The Test is Passed for given Time Frame';
        2: Status := 'The Test is Failed for given Time Frame';
        4: Status := 'Test is Running';
    END_CASE;

    END_METHOD

    (**
            Testing REAL Equality
    **)

    METHOD assertEquals

        VAR_INPUT
            IN : BOOL;
            realActualResult : REAL;
            realExpectedResult : REAL;
        END_VAR

        VAR_IN_OUT
            Status : STRING;
        END_VAR

        VAR
            Output : INT;

        END_VAR

        Init();

    IF (IN) THEN
        IF  (realActualResult = realExpectedResult) THEN
            PassTimer.IN := TRUE;

            IF(NOT PassTimer.Q) THEN
                Output := 4;
            END_IF;

            IF(PassTimer.Q) THEN
                Output := 1;
                PassTimer.IN := FALSE;

            END_IF;

        ELSIF (realActualResult <> realExpectedResult) THEN
            FailTimer(In := TRUE);

            IF(NOT FailTimer.Q) THEN
                Output := 4;
            END_IF;

            IF(FailTimer.Q) THEN
               Output := 2;
               FailTimer.In := FALSE;

            END_IF;
        END_IF;
    ELSIF (NOT IN) AND (Output<>0) THEN
                //Output := 0;

    END_IF;

    CASE Output OF
        0: Status := 'The Test is not Running';
        1: Status := 'The Test is Passed for given Time Frame';
        2: Status := 'The Test is Failed for given Time Frame';
        4: Status := 'Test is Running';
    END_CASE;

    END_METHOD

    (**
           Testing BOOLEAN Equality
    **)

    METHOD assertEquals

        VAR_INPUT
            IN : BOOL;
            boolActualResult :BOOL;
            boolExpectedResult : BOOL;

        END_VAR

        VAR_IN_OUT
            Status : STRING;
        END_VAR

        VAR
            Output : INT;

        END_VAR

        Init();

    IF (IN) THEN
        IF  (boolActualResult = boolExpectedResult) THEN
            PassTimer.IN := TRUE;

            IF(NOT PassTimer.Q) THEN
                Output := 4;
            END_IF;

            IF(PassTimer.Q) THEN
                Output := 1;
                PassTimer.IN := FALSE;
            END_IF;

        ELSIF (boolActualResult <> boolExpectedResult) THEN
            FailTimer(In := TRUE);

            IF(NOT FailTimer.Q) THEN
                Output := 4;
            END_IF;

            IF(FailTimer.Q) THEN
               Output := 2;
               FailTimer.In := FALSE;
            END_IF;
        END_IF;
    ELSIF (NOT IN) AND (Output<>0) THEN
                //Output := 0;

    END_IF;

    CASE Output OF
        0: Status := 'The Test is not Running';
        1: Status := 'The Test is Passed for given Time Frame';
        2: Status := 'The Test is Failed for given Time Frame';
        4: Status := 'Test is Running';
    END_CASE;

    END_METHOD

    METHOD assertEquals

        VAR_INPUT
            IN : BOOL;
            stringActualResult :  STRING;
            stringExpectedResult : STRING;
        END_VAR

        VAR_IN_OUT
            Status : STRING;
        END_VAR

        VAR
            Output : INT;
        END_VAR

        Init();

    IF (IN) THEN
        IF  (stringActualResult = stringExpectedResult) THEN
            PassTimer.IN := TRUE;

            IF(NOT PassTimer.Q) THEN
                Output := 4;
            END_IF;

            IF(PassTimer.Q) THEN
                Output := 1;
                PassTimer.IN := FALSE;
            END_IF;

        ELSIF (stringActualResult <> stringExpectedResult) THEN
            FailTimer(In := TRUE);

            IF(NOT FailTimer.Q) THEN
                Output := 4;
            END_IF;

            IF(FailTimer.Q) THEN
               Output := 2;
               FailTimer.In := FALSE;
            END_IF;
        END_IF;
    ELSIF (NOT IN) AND (Output<>0) THEN
                //Output := 0;

    END_IF;

    CASE Output OF
        0: Status := 'The Test is not Running';
        1: Status := 'The Test is Passed for given Time Frame';
        2: Status := 'The Test is Failed for given Time Frame';
        4: Status := 'Test is Running';
    END_CASE;

    END_METHOD

    METHOD assertTrue

        VAR_INPUT
            IN : BOOL;
            actualResult : BOOL;
        END_VAR

        VAR_IN_OUT
            Status : STRING;
        END_VAR

        VAR
            Output : INT;
        END_VAR

        Init();

    IF (IN) THEN
        IF  (actualResult = TRUE) THEN
            PassTimer.IN := TRUE;

            IF(NOT PassTimer.Q) THEN
                Output := 4;
            END_IF;

            IF(PassTimer.Q) THEN
                Output := 1;
                PassTimer.IN := FALSE;
            END_IF;

        ELSIF (actualResult = FALSE) THEN
            FailTimer(In := TRUE);

            IF(NOT FailTimer.Q) THEN
                Output := 4;
            END_IF;

            IF(FailTimer.Q) THEN
               Output := 2;
               FailTimer.In := FALSE;
            END_IF;
        END_IF;
    ELSIF (NOT IN) AND (Output<>0) THEN
                //Output := 0;

    END_IF;

    CASE Output OF
        0: Status := 'The Test is not Running';
        1: Status := 'The Test is Passed for given Time Frame';
        2: Status := 'The Test is Failed for given Time Frame';
        4: Status := 'Test is Running';
    END_CASE;

END_METHOD

    METHOD assertFalse

        VAR_INPUT
            IN : BOOL;
            actualResult : BOOL;
        END_VAR

        VAR_IN_OUT
            Status : STRING;
        END_VAR

        VAR
            Output : INT;
        END_VAR

        Init();

    IF (IN) THEN
        IF  (actualResult = FALSE) THEN
            PassTimer.IN := TRUE;

            IF(NOT PassTimer.Q) THEN
                Output := 4;
            END_IF;

            IF(PassTimer.Q) THEN
                Output := 1;
                PassTimer.IN := FALSE;
            END_IF;

        ELSIF (actualResult = TRUE) THEN
            FailTimer(In := TRUE);

            IF(NOT FailTimer.Q) THEN
                Output := 4;
            END_IF;

            IF(FailTimer.Q) THEN
               Output := 2;
               FailTimer.In := FALSE;
            END_IF;
        END_IF;
    ELSIF (NOT IN) AND (Output<>0) THEN
                //Output := 0;

    END_IF;

    CASE Output OF
        0: Status := 'The Test is not Running';
        1: Status := 'The Test is False and Passed ';
        2: Status := 'The Test is True and Failed';
        4: Status := 'Test is Running';
    END_CASE;

END_METHOD

END_CLASS
